FUNCTION TryConvert_TOD_TO_REAL : BOOL
VAR_INPUT
	in : TOD;
	out : REFERENCE TO REAL;
END_VAR

out := TOD_TO_REAL(in);
TryConvert_TOD_TO_REAL := TRUE;

END_FUNCTION

(* stored: Version 1.1.0.1, ProductVersion 3.1.4024.12
   POU TryConvert_TOD_TO_REAL: Id {734e7d22-ea80-4c8e-a660-edfd05194a62}, SpecialFunc None *)
